{attribute 'GeneratedUsingTerminal: EK1501-0000-0016'}
{attribute addProperty BoxType "EK1501-0000-0016"}
{attribute addProperty Id "EtcSlaveTerminalBaseIDAT %I*ID_07C9D28F2WcStateAT %I*WcState_9091E0EB2InfoDataAT %I*InfoData_6F19DB2B2"}
{attribute addProperty CRC "3382454092"}
{attribute addProperty Size "6"}
TYPE EK1501_C99C274C EXTENDS EtcSlaveTerminalBase :
STRUCT
	{attribute addProperty Name "ID"}
	ID : ID_07C9D28F;
	{attribute addProperty Name "WcState"}
	WcState : WcState_9091E0EB;
	{attribute addProperty Name "InfoData"}
	InfoData : InfoData_6F19DB2B;
END_STRUCT
END_TYPE

(* stored: Version 1.2.0.0, ProductVersion 3.1.4024.9
   DUT EK1501_C99C274C: Id {8497a98c-54a8-4c16-869f-3ca70f808ada} *)
